TYPE ST_DataExchange : 
	STRUCT
	
		Dynamics : ST_Dynamics;
		Reset : BOOL;
		Run : BOOL;
		SafetyInRun : BOOL;
		{attribute 'hide'}
		_reserved1 : ARRAY [1..5] OF USINT;
	END_STRUCT
END_TYPE

(* stored: Version 1.1.0.1, ProductVersion 3.1.4026.8
   DUT ST_DataExchange: Id {80b78fb9-86bf-4f62-8cb9-2fe377a6eb18} *)
